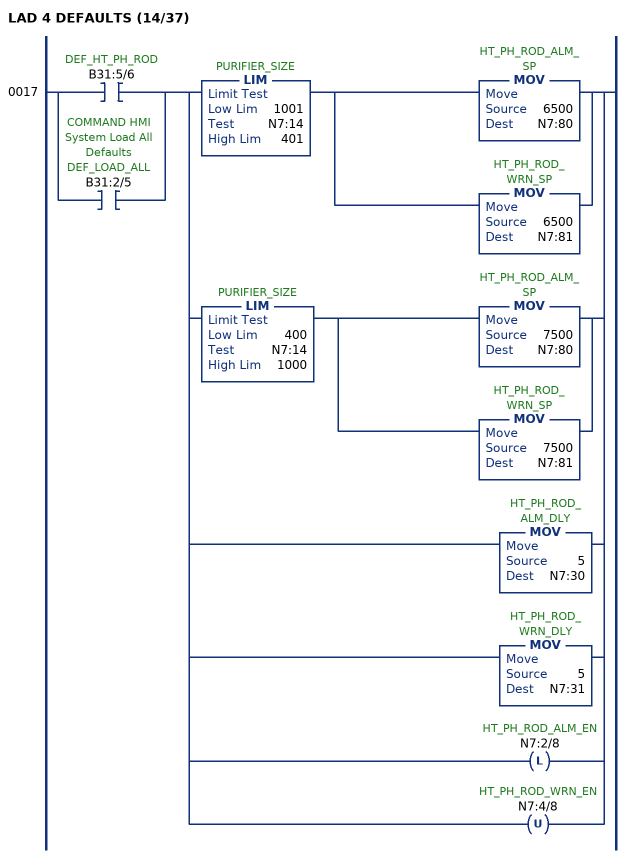
% Rung: 17 %
SOR BST XIC B31:5/6 NXB XIC B31:2/5 BND BST LIM 1001 N7:14 401 BST MOV 6500 N7:80 NXB MOV 6500 N7:81 BND NXB LIM 400 N7:14 1000 BST MOV 7500 N7:80 NXB MOV 7500 N7:81 BND NXB MOV 5 N7:30 NXB MOV 5 N7:31 NXB OTL N7:2/8 NXB OTU N7:4/8 BND EOR
%   B31:5/6  DEF_HT_PH_ROD %
%   B31:2/5  DEF_LOAD_ALL  "COMMAND HMI System Load All Defaults" %
%   N7:14  PURIFIER_SIZE %
%   N7:80  HT_PH_ROD_ALM_SP %
%   N7:81  HT_PH_ROD_WRN_SP %
%   N7:30  HT_PH_ROD_ALM_DLY %
%   N7:31  HT_PH_ROD_WRN_DLY %
%   N7:2/8  HT_PH_ROD_ALM_EN %
%   N7:4/8  HT_PH_ROD_WRN_EN %

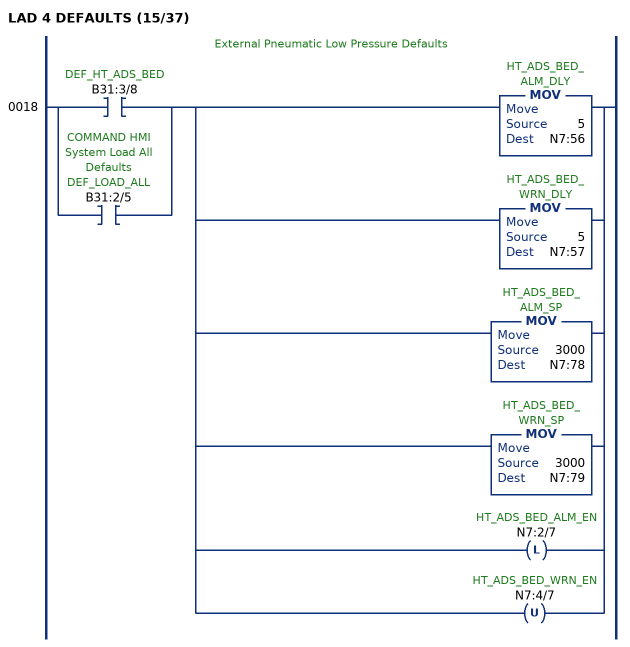
% Rung: 18 %
% External Pneumatic Low Pressure Defaults %
SOR BST XIC B31:3/8 NXB XIC B31:2/5 BND BST MOV 5 N7:56 NXB MOV 5 N7:57 NXB MOV 3000 N7:78 NXB MOV 3000 N7:79 NXB OTL N7:2/7 NXB OTU N7:4/7 BND EOR
%   B31:3/8  DEF_HT_ADS_BED %
%   B31:2/5  DEF_LOAD_ALL  "COMMAND HMI System Load All Defaults" %
%   N7:56  HT_ADS_BED_ALM_DLY %
%   N7:57  HT_ADS_BED_WRN_DLY %
%   N7:78  HT_ADS_BED_ALM_SP %
%   N7:79  HT_ADS_BED_WRN_SP %
%   N7:2/7  HT_ADS_BED_ALM_EN %
%   N7:4/7  HT_ADS_BED_WRN_EN %

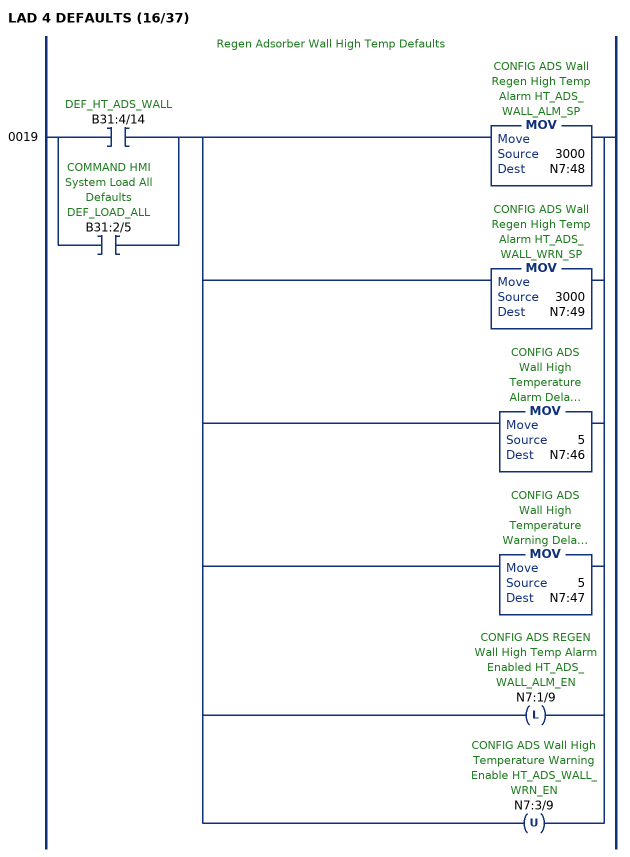
% Rung: 19 %
% Regen Adsorber Wall High Temp Defaults %
SOR BST XIC B31:4/14 NXB XIC B31:2/5 BND BST BST MOV 3000 N7:48 NXB MOV 3000 N7:49 BND NXB MOV 5 N7:46 NXB MOV 5 N7:47 NXB OTL N7:1/9 NXB OTU N7:3/9 BND EOR
%   B31:4/14  DEF_HT_ADS_WALL %
%   B31:2/5  DEF_LOAD_ALL  "COMMAND HMI System Load All Defaults" %
%   N7:48  HT_ADS_WALL_ALM_SP  "CONFIG ADS Wall Regen High Temp Alarm" %
%   N7:49  HT_ADS_WALL_WRN_SP  "CONFIG ADS Wall Regen High Temp Alarm" %
%   N7:46  HT_ADS_WALL_ALM_DLY  "CONFIG ADS Wall High Temperature Alarm Delay" %
%   N7:47  HT_ADS_WALL_WRN_DLY  "CONFIG ADS Wall High Temperature Warning Delay" %
%   N7:1/9  HT_ADS_WALL_ALM_EN  "CONFIG ADS REGEN Wall High Temp Alarm Enabled" %
%   N7:3/9  HT_ADS_WALL_WRN_EN  "CONFIG ADS Wall High Temperature Warning Enable" %

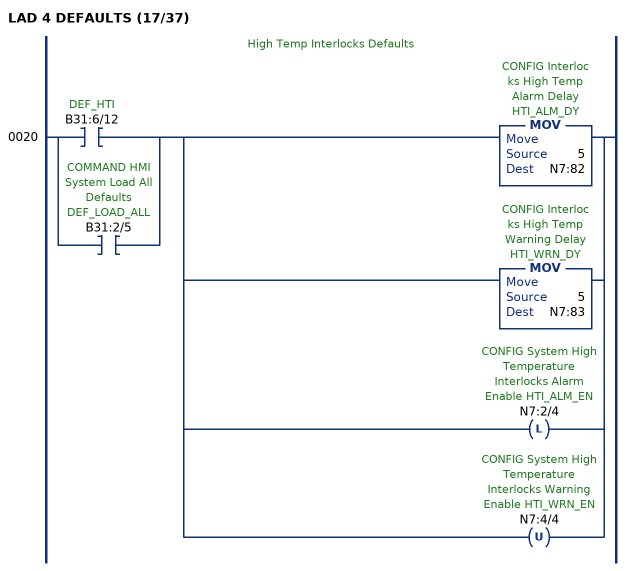
% Rung: 20 %
% High Temp Interlocks Defaults %
SOR BST XIC B31:6/12 NXB XIC B31:2/5 BND BST MOV 5 N7:82 NXB MOV 5 N7:83 NXB OTL N7:2/4 NXB OTU N7:4/4 BND EOR
%   B31:6/12  DEF_HTI %
%   B31:2/5  DEF_LOAD_ALL  "COMMAND HMI System Load All Defaults" %
%   N7:82  HTI_ALM_DY  "CONFIG Interlocks High Temp Alarm Delay" %
%   N7:83  HTI_WRN_DY  "CONFIG Interlocks High Temp Warning Delay" %
%   N7:2/4  HTI_ALM_EN  "CONFIG System High Temperature Interlocks Alarm Enable" %
%   N7:4/4  HTI_WRN_EN  "CONFIG System High Temperature Interlocks Warning Enable" %

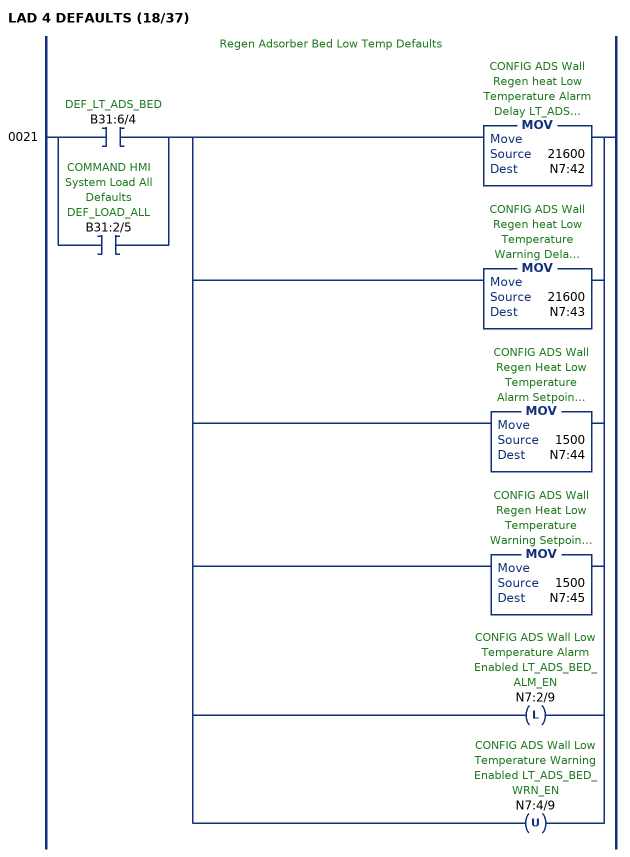
% Rung: 21 %
% Regen Adsorber Bed Low Temp Defaults %
SOR BST XIC B31:6/4 NXB XIC B31:2/5 BND BST MOV 21600 N7:42 NXB MOV 21600 N7:43 NXB MOV 1500 N7:44 NXB MOV 1500 N7:45 NXB OTL N7:2/9 NXB OTU N7:4/9 BND EOR
%   B31:6/4  DEF_LT_ADS_BED %
%   B31:2/5  DEF_LOAD_ALL  "COMMAND HMI System Load All Defaults" %
%   N7:42  LT_ADS_BED_ALM_DLY  "CONFIG ADS Wall Regen heat Low Temperature Alarm Delay" %
%   N7:43  LT_ADS_BED_WRN_DLY  "CONFIG ADS Wall Regen heat Low Temperature Warning Delay" %
%   N7:44  LT_ADS_BED_ALM_SP  "CONFIG ADS Wall Regen Heat Low Temperature Alarm Setpoint" %
%   N7:45  LT_ADS_BED_WRN_SP  "CONFIG ADS Wall Regen Heat Low Temperature Warning Setpoint" %
%   N7:2/9  LT_ADS_BED_ALM_EN  "CONFIG ADS Wall Low Temperature Alarm Enabled" %
%   N7:4/9  LT_ADS_BED_WRN_EN  "CONFIG ADS Wall Low Temperature Warning Enabled" %

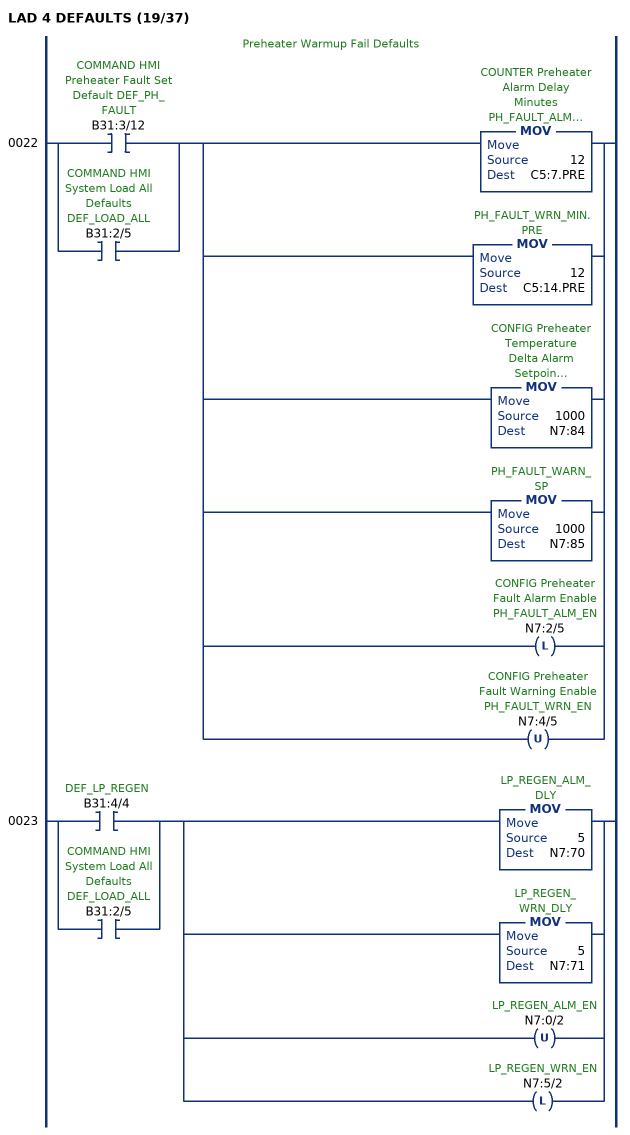
% Rung: 22 %
% Preheater Warmup Fail Defaults %
SOR BST XIC B31:3/12 NXB XIC B31:2/5 BND BST MOV 12 C5:7.PRE NXB MOV 12 C5:14.PRE NXB MOV 1000 N7:84 NXB MOV 1000 N7:85 NXB OTL N7:2/5 NXB OTU N7:4/5 BND EOR
%   B31:3/12  DEF_PH_FAULT  "COMMAND HMI Preheater Fault Set Default" %
%   B31:2/5  DEF_LOAD_ALL  "COMMAND HMI System Load All Defaults" %
%   C5:7  PH_FAULT_ALM_MIN  "COUNTER Preheater Alarm Delay Minutes" %
%   C5:14  PH_FAULT_WRN_MIN %
%   N7:84  PH_FAULT_ALARM_SP  "CONFIG Preheater Temperature Delta Alarm Setpoint" %
%   N7:85  PH_FAULT_WARN_SP %
%   N7:2/5  PH_FAULT_ALM_EN  "CONFIG Preheater Fault Alarm Enable" %
%   N7:4/5  PH_FAULT_WRN_EN  "CONFIG Preheater Fault Warning Enable" %
% Rung: 23 %
SOR BST XIC B31:4/4 NXB XIC B31:2/5 BND BST MOV 5 N7:70 NXB MOV 5 N7:71 NXB OTU N7:0/2 NXB OTL N7:5/2 BND EOR
%   B31:4/4  DEF_LP_REGEN %
%   B31:2/5  DEF_LOAD_ALL  "COMMAND HMI System Load All Defaults" %
%   N7:70  LP_REGEN_ALM_DLY %
%   N7:71  LP_REGEN_WRN_DLY %
%   N7:0/2  LP_REGEN_ALM_EN %
%   N7:5/2  LP_REGEN_WRN_EN %

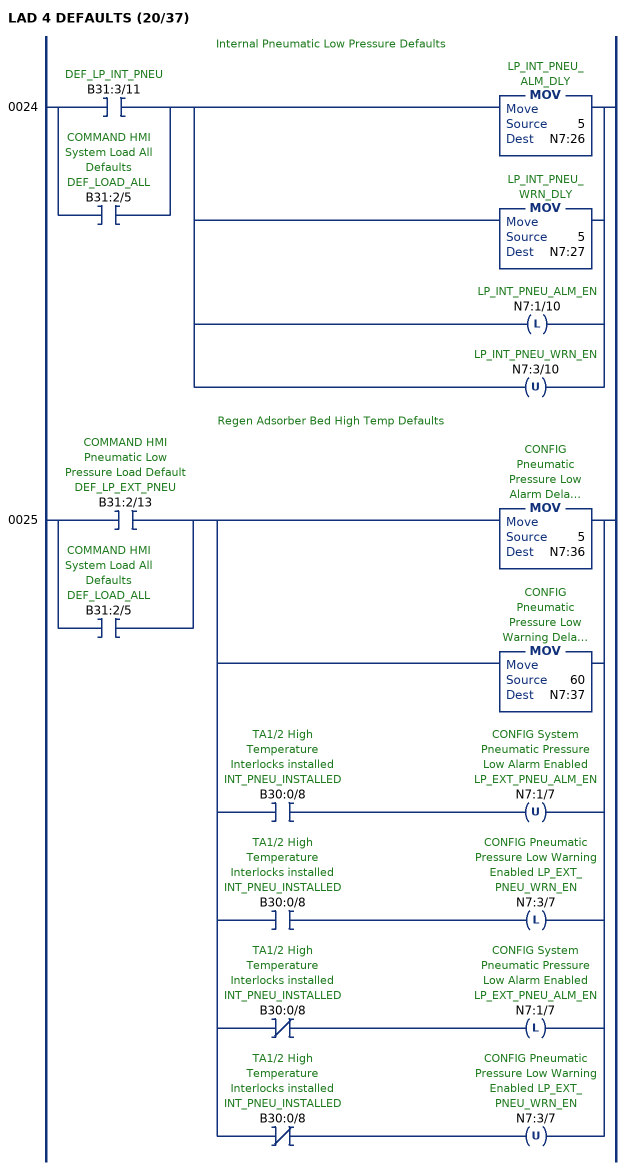
% Rung: 24 %
% Internal Pneumatic Low Pressure Defaults %
SOR BST XIC B31:3/11 NXB XIC B31:2/5 BND BST MOV 5 N7:26 NXB MOV 5 N7:27 NXB OTL N7:1/10 NXB OTU N7:3/10 BND EOR
%   B31:3/11  DEF_LP_INT_PNEU %
%   B31:2/5  DEF_LOAD_ALL  "COMMAND HMI System Load All Defaults" %
%   N7:26  LP_INT_PNEU_ALM_DLY %
%   N7:27  LP_INT_PNEU_WRN_DLY %
%   N7:1/10  LP_INT_PNEU_ALM_EN %
%   N7:3/10  LP_INT_PNEU_WRN_EN %
% Rung: 25 %
% Regen Adsorber Bed High Temp Defaults %
SOR BST XIC B31:2/13 NXB XIC B31:2/5 BND BST MOV 5 N7:36 NXB MOV 60 N7:37 NXB XIC B30:0/8 OTU N7:1/7 NXB XIC B30:0/8 OTL N7:3/7 NXB XIO B30:0/8 OTL N7:1/7 NXB XIO B30:0/8 OTU N7:3/7 BND EOR
%   B31:2/13  DEF_LP_EXT_PNEU  "COMMAND HMI Pneumatic Low Pressure Load Default" %
%   B31:2/5  DEF_LOAD_ALL  "COMMAND HMI System Load All Defaults" %
%   N7:36  LP_EXT_PNEU_ALM_DLY  "CONFIG Pneumatic Pressure Low Alarm Delay" %
%   N7:37  LP_EXT_PNEU_WRN_DLY  "CONFIG Pneumatic Pressure Low Warning Delay" %
%   B30:0/8  INT_PNEU_INSTALLED  "TA1/2 High Temperature Interlocks installed" %
%   N7:1/7  LP_EXT_PNEU_ALM_EN  "CONFIG System Pneumatic Pressure Low Alarm Enabled" %
%   N7:3/7  LP_EXT_PNEU_WRN_EN  "CONFIG Pneumatic Pressure Low Warning Enabled" %

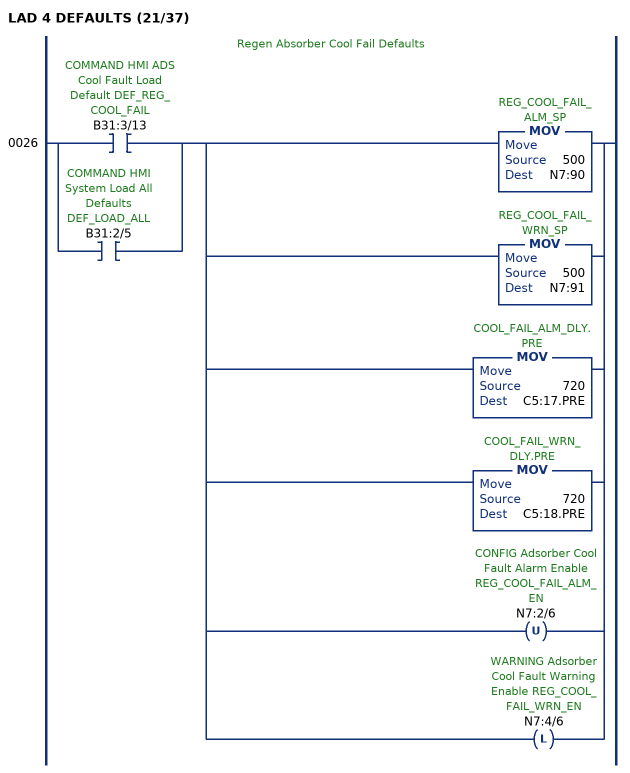
% Rung: 26 %
% Regen Absorber Cool Fail Defaults %
SOR BST XIC B31:3/13 NXB XIC B31:2/5 BND BST MOV 500 N7:90 NXB MOV 500 N7:91 NXB MOV 720 C5:17.PRE NXB MOV 720 C5:18.PRE NXB OTU N7:2/6 NXB OTL N7:4/6 BND EOR
%   B31:3/13  DEF_REG_COOL_FAIL  "COMMAND HMI ADS Cool Fault Load Default" %
%   B31:2/5  DEF_LOAD_ALL  "COMMAND HMI System Load All Defaults" %
%   N7:90  REG_COOL_FAIL_ALM_SP %
%   N7:91  REG_COOL_FAIL_WRN_SP %
%   C5:17  COOL_FAIL_ALM_DLY %
%   C5:18  COOL_FAIL_WRN_DLY %
%   N7:2/6  REG_COOL_FAIL_ALM_EN  "CONFIG Adsorber Cool Fault Alarm Enable" %
%   N7:4/6  REG_COOL_FAIL_WRN_EN  "WARNING Adsorber Cool Fault Warning Enable" %

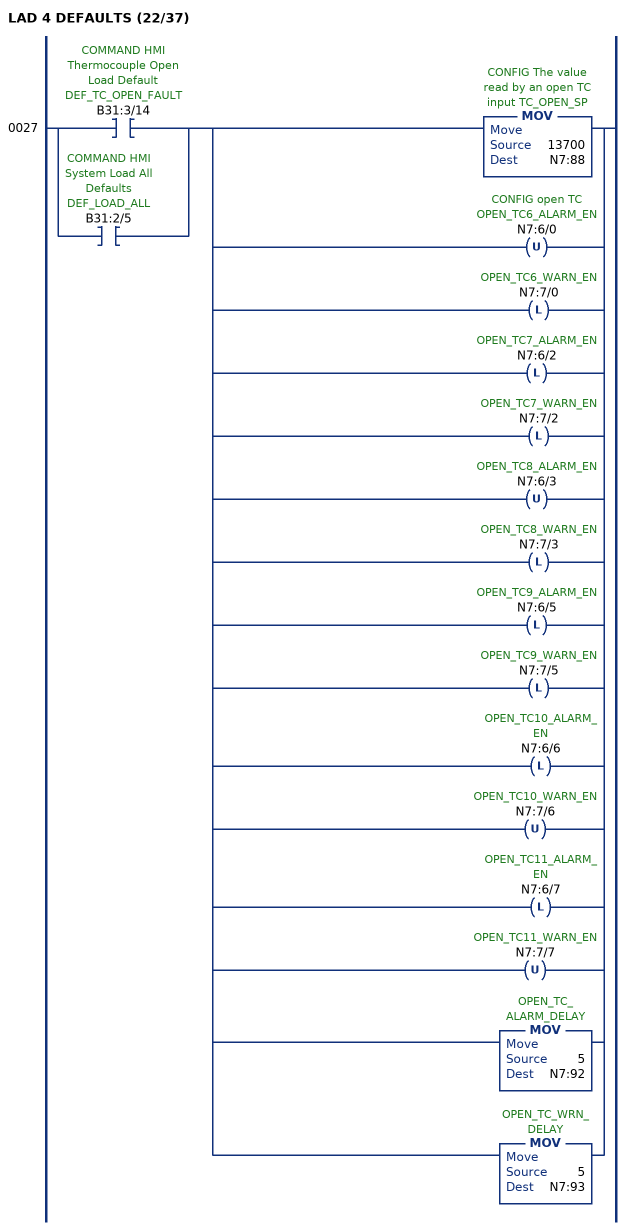
% Rung: 27 %
SOR BST XIC B31:3/14 NXB XIC B31:2/5 BND BST MOV 13700 N7:88 NXB OTU N7:6/0 NXB OTL N7:7/0 NXB OTL N7:6/2 NXB OTL N7:7/2 NXB OTU N7:6/3 NXB OTL N7:7/3 NXB OTL N7:6/5 NXB OTL N7:7/5 NXB OTL N7:6/6 NXB OTU N7:7/6 NXB OTL N7:6/7 NXB BST OTU N7:7/7 NXB BST MOV 5 N7:92 NXB MOV 5 N7:93 BND BND BND EOR
%   B31:3/14  DEF_TC_OPEN_FAULT  "COMMAND HMI Thermocouple Open Load Default" %
%   B31:2/5  DEF_LOAD_ALL  "COMMAND HMI System Load All Defaults" %
%   N7:88  TC_OPEN_SP  "CONFIG The value read by an open TC input" %
%   N7:6/0  OPEN_TC6_ALARM_EN  "CONFIG open TC" %
%   N7:7/0  OPEN_TC6_WARN_EN %
%   N7:6/2  OPEN_TC7_ALARM_EN %
%   N7:7/2  OPEN_TC7_WARN_EN %
%   N7:6/3  OPEN_TC8_ALARM_EN %
%   N7:7/3  OPEN_TC8_WARN_EN %
%   N7:6/5  OPEN_TC9_ALARM_EN %
%   N7:7/5  OPEN_TC9_WARN_EN %
%   N7:6/6  OPEN_TC10_ALARM_EN %
%   N7:7/6  OPEN_TC10_WARN_EN %
%   N7:6/7  OPEN_TC11_ALARM_EN %
%   N7:7/7  OPEN_TC11_WARN_EN %
%   N7:92  OPEN_TC_ALARM_DELAY %
%   N7:93  OPEN_TC_WRN_DELAY %

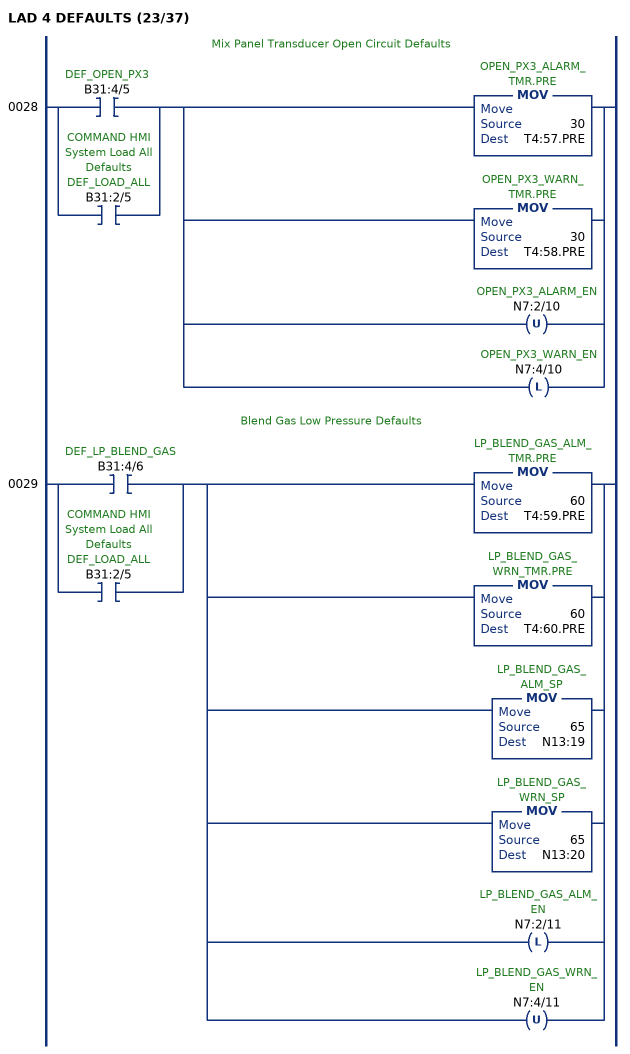
% Rung: 28 %
% Mix Panel Transducer Open Circuit Defaults %
SOR BST XIC B31:4/5 NXB XIC B31:2/5 BND BST MOV 30 T4:57.PRE NXB MOV 30 T4:58.PRE NXB OTU N7:2/10 NXB OTL N7:4/10 BND EOR
%   B31:4/5  DEF_OPEN_PX3 %
%   B31:2/5  DEF_LOAD_ALL  "COMMAND HMI System Load All Defaults" %
%   T4:57  OPEN_PX3_ALARM_TMR %
%   T4:58  OPEN_PX3_WARN_TMR %
%   N7:2/10  OPEN_PX3_ALARM_EN %
%   N7:4/10  OPEN_PX3_WARN_EN %
% Rung: 29 %
% Blend Gas Low Pressure Defaults %
SOR BST XIC B31:4/6 NXB XIC B31:2/5 BND BST MOV 60 T4:59.PRE NXB MOV 60 T4:60.PRE NXB MOV 65 N13:19 NXB MOV 65 N13:20 NXB OTL N7:2/11 NXB OTU N7:4/11 BND EOR
%   B31:4/6  DEF_LP_BLEND_GAS %
%   B31:2/5  DEF_LOAD_ALL  "COMMAND HMI System Load All Defaults" %
%   T4:59  LP_BLEND_GAS_ALM_TMR %
%   T4:60  LP_BLEND_GAS_WRN_TMR %
%   N13:19  LP_BLEND_GAS_ALM_SP %
%   N13:20  LP_BLEND_GAS_WRN_SP %
%   N7:2/11  LP_BLEND_GAS_ALM_EN %
%   N7:4/11  LP_BLEND_GAS_WRN_EN %

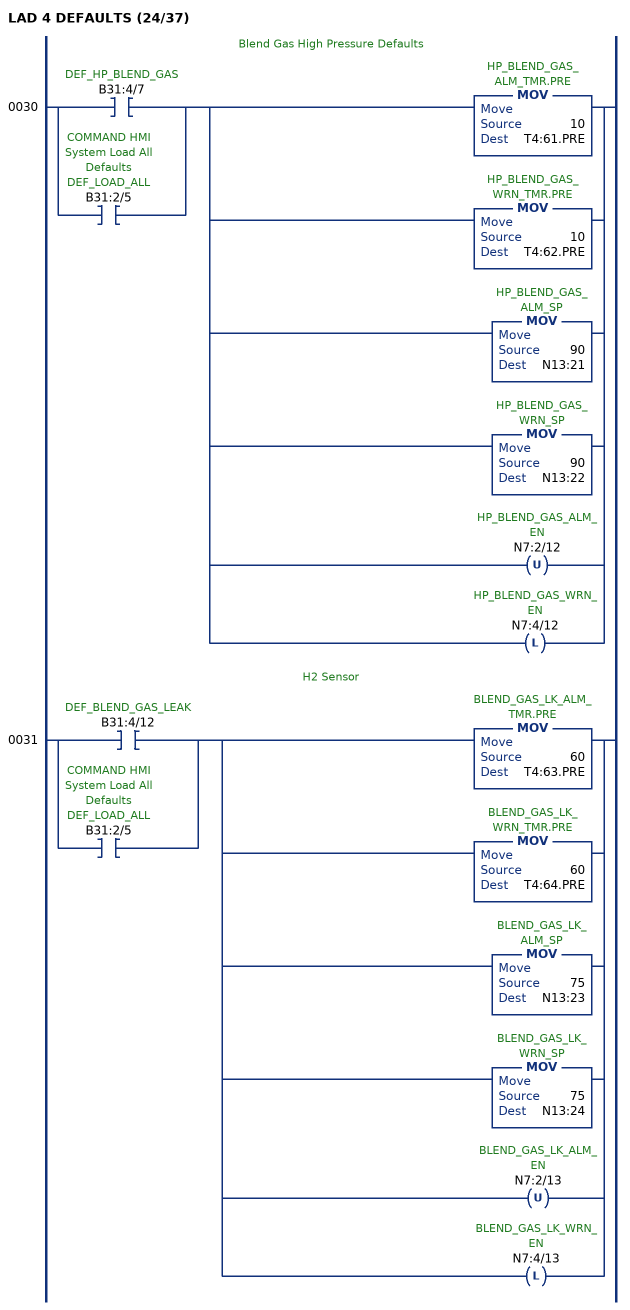
% Rung: 30 %
% Blend Gas High Pressure Defaults %
SOR BST XIC B31:4/7 NXB XIC B31:2/5 BND BST MOV 10 T4:61.PRE NXB MOV 10 T4:62.PRE NXB MOV 90 N13:21 NXB MOV 90 N13:22 NXB OTU N7:2/12 NXB OTL N7:4/12 BND EOR
%   B31:4/7  DEF_HP_BLEND_GAS %
%   B31:2/5  DEF_LOAD_ALL  "COMMAND HMI System Load All Defaults" %
%   T4:61  HP_BLEND_GAS_ALM_TMR %
%   T4:62  HP_BLEND_GAS_WRN_TMR %
%   N13:21  HP_BLEND_GAS_ALM_SP %
%   N13:22  HP_BLEND_GAS_WRN_SP %
%   N7:2/12  HP_BLEND_GAS_ALM_EN %
%   N7:4/12  HP_BLEND_GAS_WRN_EN %
% Rung: 31 %
% H2 Sensor %
SOR BST XIC B31:4/12 NXB XIC B31:2/5 BND BST MOV 60 T4:63.PRE NXB MOV 60 T4:64.PRE NXB MOV 75 N13:23 NXB MOV 75 N13:24 NXB OTU N7:2/13 NXB OTL N7:4/13 BND EOR
%   B31:4/12  DEF_BLEND_GAS_LEAK %
%   B31:2/5  DEF_LOAD_ALL  "COMMAND HMI System Load All Defaults" %
%   T4:63  BLEND_GAS_LK_ALM_TMR %
%   T4:64  BLEND_GAS_LK_WRN_TMR %
%   N13:23  BLEND_GAS_LK_ALM_SP %
%   N13:24  BLEND_GAS_LK_WRN_SP %
%   N7:2/13  BLEND_GAS_LK_ALM_EN %
%   N7:4/13  BLEND_GAS_LK_WRN_EN %

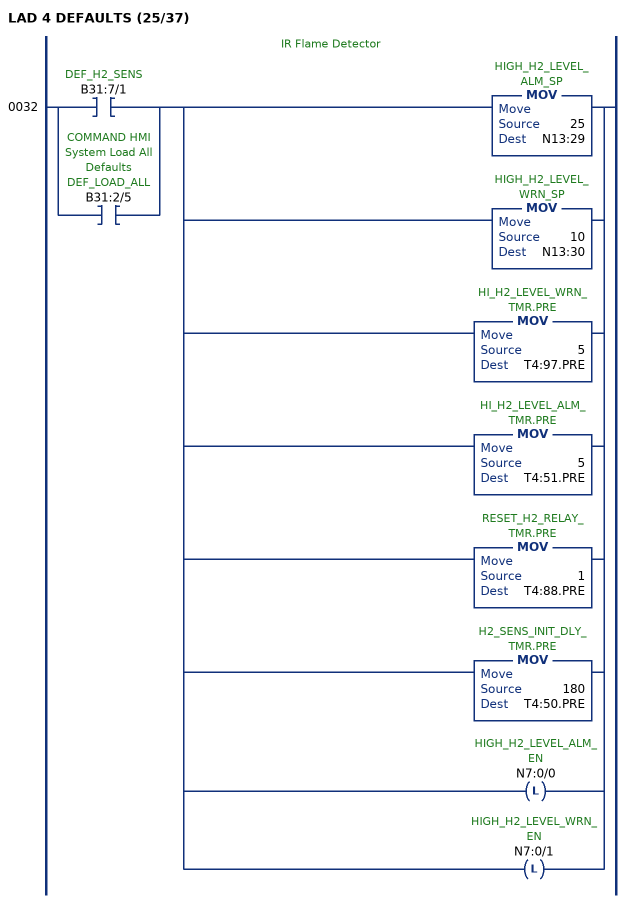
% Rung: 32 %
% IR Flame Detector %
SOR BST XIC B31:7/1 NXB XIC B31:2/5 BND BST MOV 25 N13:29 NXB MOV 10 N13:30 NXB MOV 5 T4:97.PRE NXB MOV 5 T4:51.PRE NXB MOV 1 T4:88.PRE NXB MOV 180 T4:50.PRE NXB OTL N7:0/0 NXB OTL N7:0/1 BND EOR
%   B31:7/1  DEF_H2_SENS %
%   B31:2/5  DEF_LOAD_ALL  "COMMAND HMI System Load All Defaults" %
%   N13:29  HIGH_H2_LEVEL_ALM_SP %
%   N13:30  HIGH_H2_LEVEL_WRN_SP %
%   T4:97  HI_H2_LEVEL_WRN_TMR %
%   T4:51  HI_H2_LEVEL_ALM_TMR %
%   T4:88  RESET_H2_RELAY_TMR %
%   T4:50  H2_SENS_INIT_DLY_TMR %
%   N7:0/0  HIGH_H2_LEVEL_ALM_EN %
%   N7:0/1  HIGH_H2_LEVEL_WRN_EN %

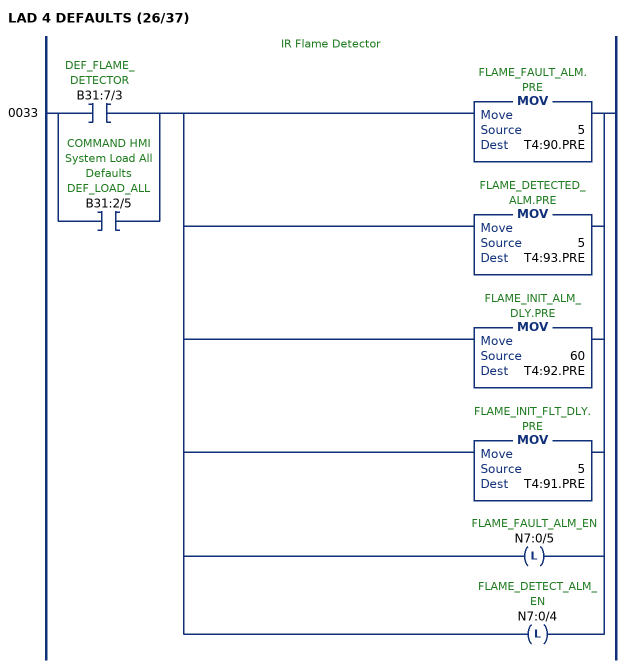
% Rung: 33 %
% IR Flame Detector %
SOR BST XIC B31:7/3 NXB XIC B31:2/5 BND BST MOV 5 T4:90.PRE NXB MOV 5 T4:93.PRE NXB MOV 60 T4:92.PRE NXB MOV 5 T4:91.PRE NXB OTL N7:0/5 NXB OTL N7:0/4 BND EOR
%   B31:7/3  DEF_FLAME_DETECTOR %
%   B31:2/5  DEF_LOAD_ALL  "COMMAND HMI System Load All Defaults" %
%   T4:90  FLAME_FAULT_ALM %
%   T4:93  FLAME_DETECTED_ALM %
%   T4:92  FLAME_INIT_ALM_DLY %
%   T4:91  FLAME_INIT_FLT_DLY %
%   N7:0/5  FLAME_FAULT_ALM_EN %
%   N7:0/4  FLAME_DETECT_ALM_EN %

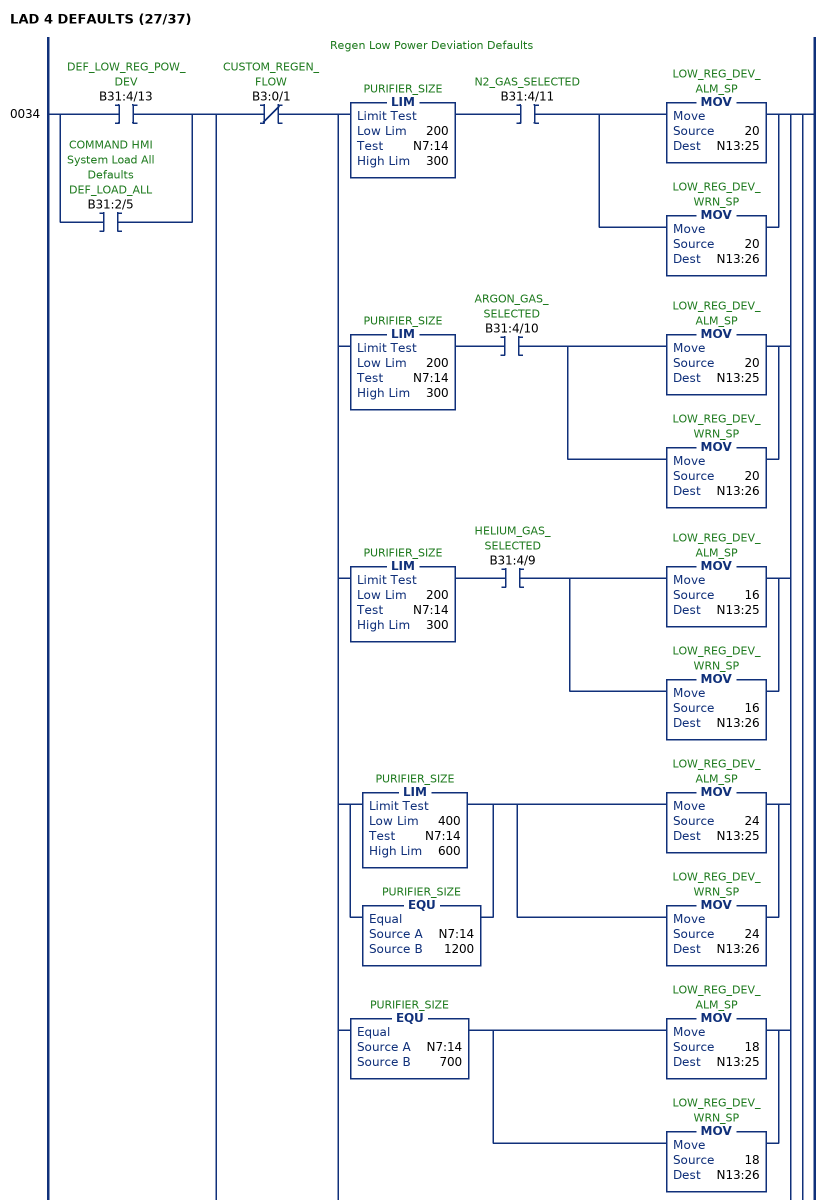

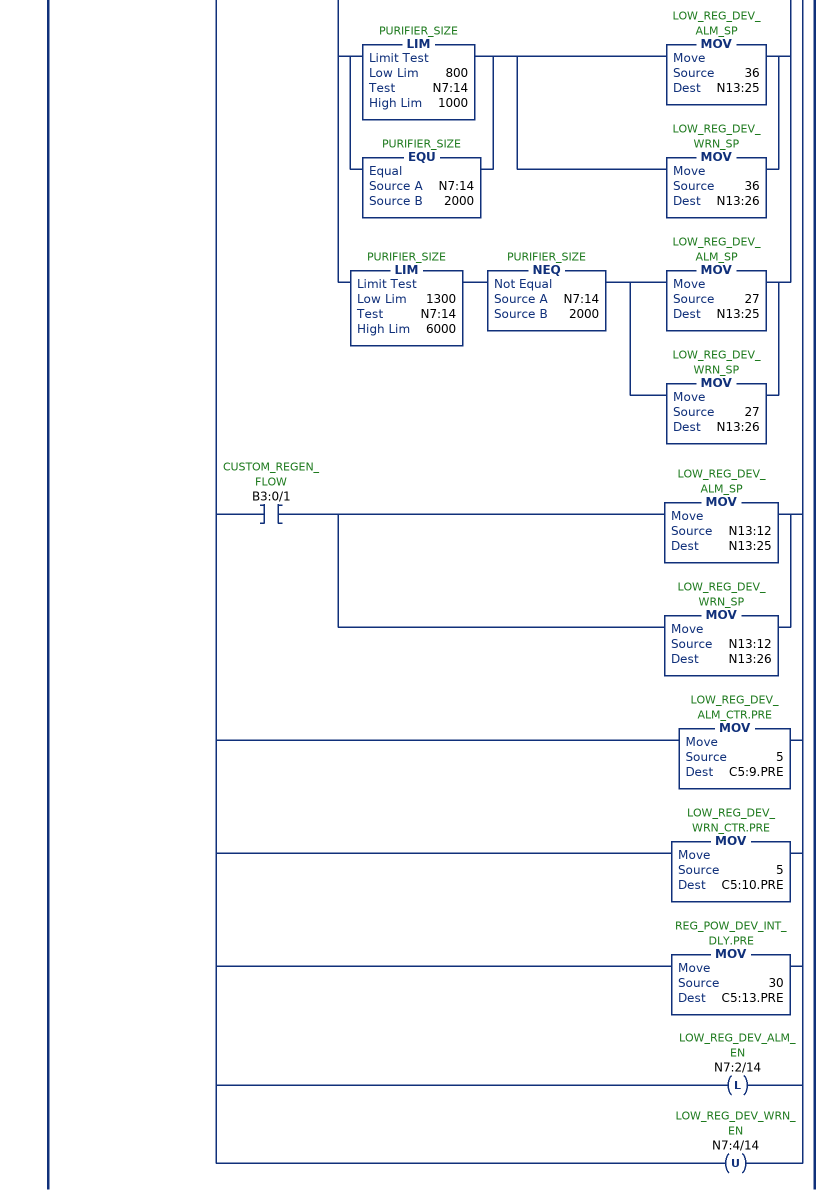
% Rung: 34 %
% Regen Low Power Deviation Defaults %
SOR BST XIC B31:4/13 NXB XIC B31:2/5 BND BST XIO B3:0/1 BST LIM 200 N7:14 300 XIC B31:4/11 BST MOV 20 N13:25 NXB MOV 20 N13:26 BND NXB LIM 200 N7:14 300 XIC B31:4/10 BST MOV 20 N13:25 NXB MOV 20 N13:26 BND NXB LIM 200 N7:14 300 XIC B31:4/9 BST MOV 16 N13:25 NXB MOV 16 N13:26 BND NXB BST LIM 400 N7:14 600 NXB EQU N7:14 1200 BND BST MOV 24 N13:25 NXB MOV 24 N13:26 BND NXB EQU N7:14 700 BST MOV 18 N13:25 NXB MOV 18 N13:26 BND NXB BST LIM 800 N7:14 1000 NXB EQU N7:14 2000 BND BST MOV 36 N13:25 NXB MOV 36 N13:26 BND NXB LIM 1300 N7:14 6000 NEQ N7:14 2000 BST MOV 27 N13:25 NXB MOV 27 N13:26 BND BND NXB XIC B3:0/1 BST MOV N13:12 N13:25 NXB MOV N13:12 N13:26 BND NXB MOV 5 C5:9.PRE NXB MOV 5 C5:10.PRE NXB MOV 30 C5:13.PRE NXB OTL N7:2/14 NXB OTU N7:4/14 BND EOR
%   B31:4/13  DEF_LOW_REG_POW_DEV %
%   B31:2/5  DEF_LOAD_ALL  "COMMAND HMI System Load All Defaults" %
%   B3:0/1  CUSTOM_REGEN_FLOW %
%   N7:14  PURIFIER_SIZE %
%   B31:4/11  N2_GAS_SELECTED %
%   N13:25  LOW_REG_DEV_ALM_SP %
%   N13:26  LOW_REG_DEV_WRN_SP %
%   B31:4/10  ARGON_GAS_SELECTED %
%   B31:4/9  HELIUM_GAS_SELECTED %
%   N13:12  CUST_LOW_REG_DEV_SP %
%   C5:9  LOW_REG_DEV_ALM_CTR %
%   C5:10  LOW_REG_DEV_WRN_CTR %
%   C5:13  REG_POW_DEV_INT_DLY %
%   N7:2/14  LOW_REG_DEV_ALM_EN %
%   N7:4/14  LOW_REG_DEV_WRN_EN %

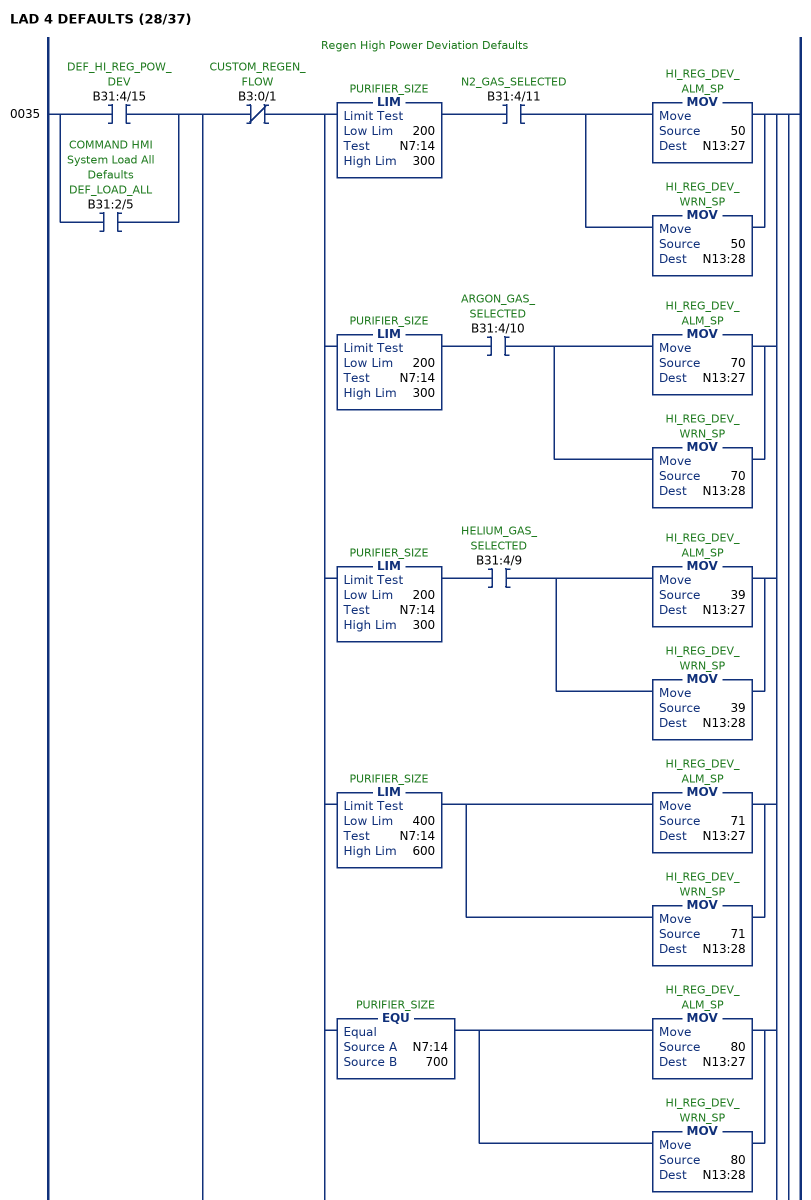

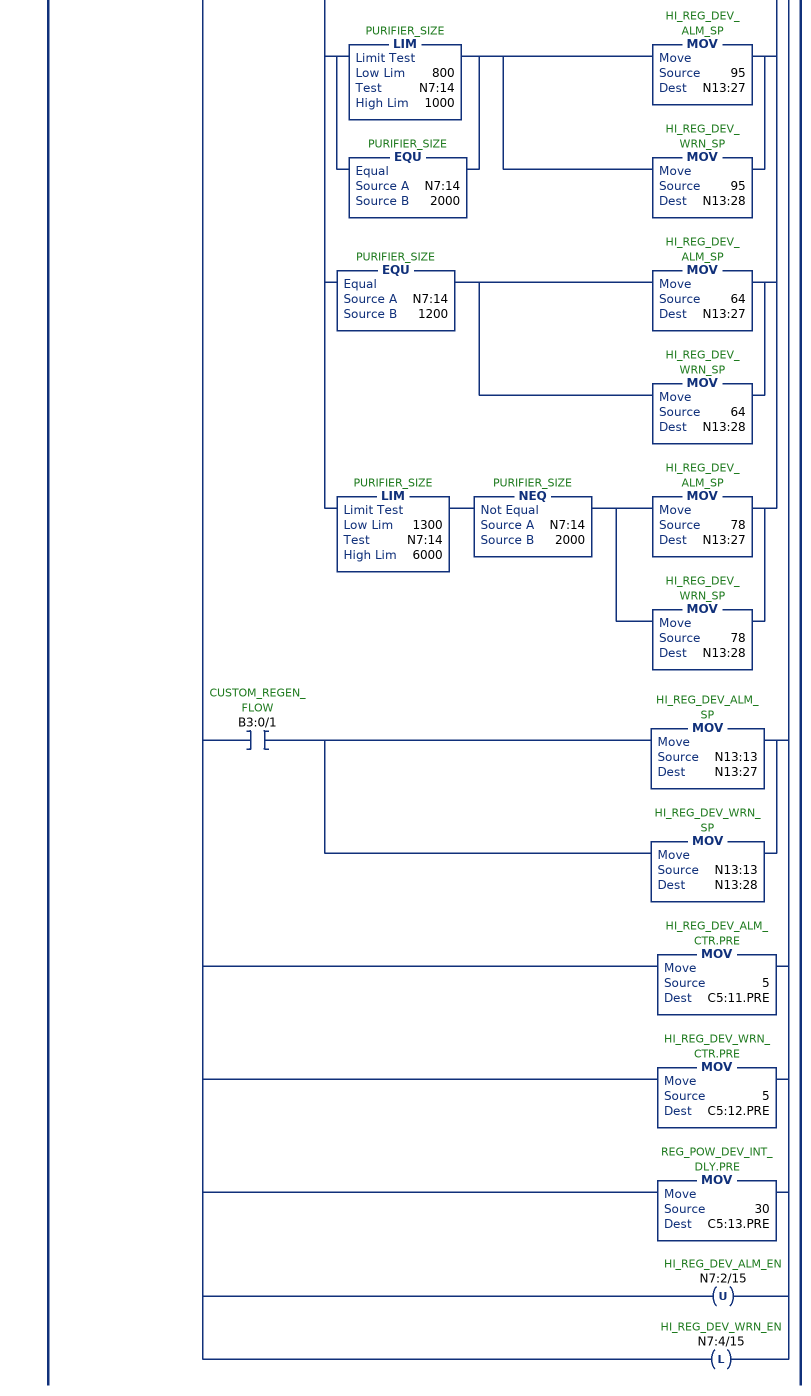
% Rung: 35 %
% Regen High Power Deviation Defaults %
SOR BST XIC B31:4/15 NXB XIC B31:2/5 BND BST XIO B3:0/1 BST LIM 200 N7:14 300 XIC B31:4/11 BST MOV 50 N13:27 NXB MOV 50 N13:28 BND NXB LIM 200 N7:14 300 XIC B31:4/10 BST MOV 70 N13:27 NXB MOV 70 N13:28 BND NXB LIM 200 N7:14 300 XIC B31:4/9 BST MOV 39 N13:27 NXB MOV 39 N13:28 BND NXB LIM 400 N7:14 600 BST MOV 71 N13:27 NXB MOV 71 N13:28 BND NXB EQU N7:14 700 BST MOV 80 N13:27 NXB MOV 80 N13:28 BND NXB BST LIM 800 N7:14 1000 NXB EQU N7:14 2000 BND BST MOV 95 N13:27 NXB MOV 95 N13:28 BND NXB EQU N7:14 1200 BST MOV 64 N13:27 NXB MOV 64 N13:28 BND NXB LIM 1300 N7:14 6000 NEQ N7:14 2000 BST MOV 78 N13:27 NXB MOV 78 N13:28 BND BND NXB XIC B3:0/1 BST MOV N13:13 N13:27 NXB MOV N13:13 N13:28 BND NXB MOV 5 C5:11.PRE NXB MOV 5 C5:12.PRE NXB MOV 30 C5:13.PRE NXB OTU N7:2/15 NXB OTL N7:4/15 BND EOR
%   B31:4/15  DEF_HI_REG_POW_DEV %
%   B31:2/5  DEF_LOAD_ALL  "COMMAND HMI System Load All Defaults" %
%   B3:0/1  CUSTOM_REGEN_FLOW %
%   N7:14  PURIFIER_SIZE %
%   B31:4/11  N2_GAS_SELECTED %
%   N13:27  HI_REG_DEV_ALM_SP %
%   N13:28  HI_REG_DEV_WRN_SP %
%   B31:4/10  ARGON_GAS_SELECTED %
%   B31:4/9  HELIUM_GAS_SELECTED %
%   N13:13  CUST_HI_REG_DEV_SP %
%   C5:11  HI_REG_DEV_ALM_CTR %
%   C5:12  HI_REG_DEV_WRN_CTR %
%   C5:13  REG_POW_DEV_INT_DLY %
%   N7:2/15  HI_REG_DEV_ALM_EN %
%   N7:4/15  HI_REG_DEV_WRN_EN %

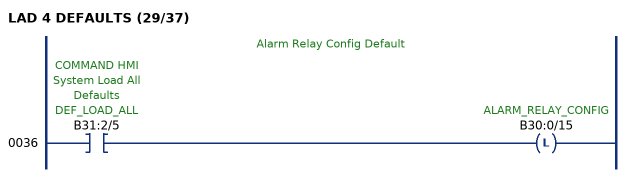
% Rung: 36 %
% Alarm Relay Config Default %
SOR XIC B31:2/5 OTL B30:0/15 EOR
%   B31:2/5  DEF_LOAD_ALL  "COMMAND HMI System Load All Defaults" %
%   B30:0/15  ALARM_RELAY_CONFIG %

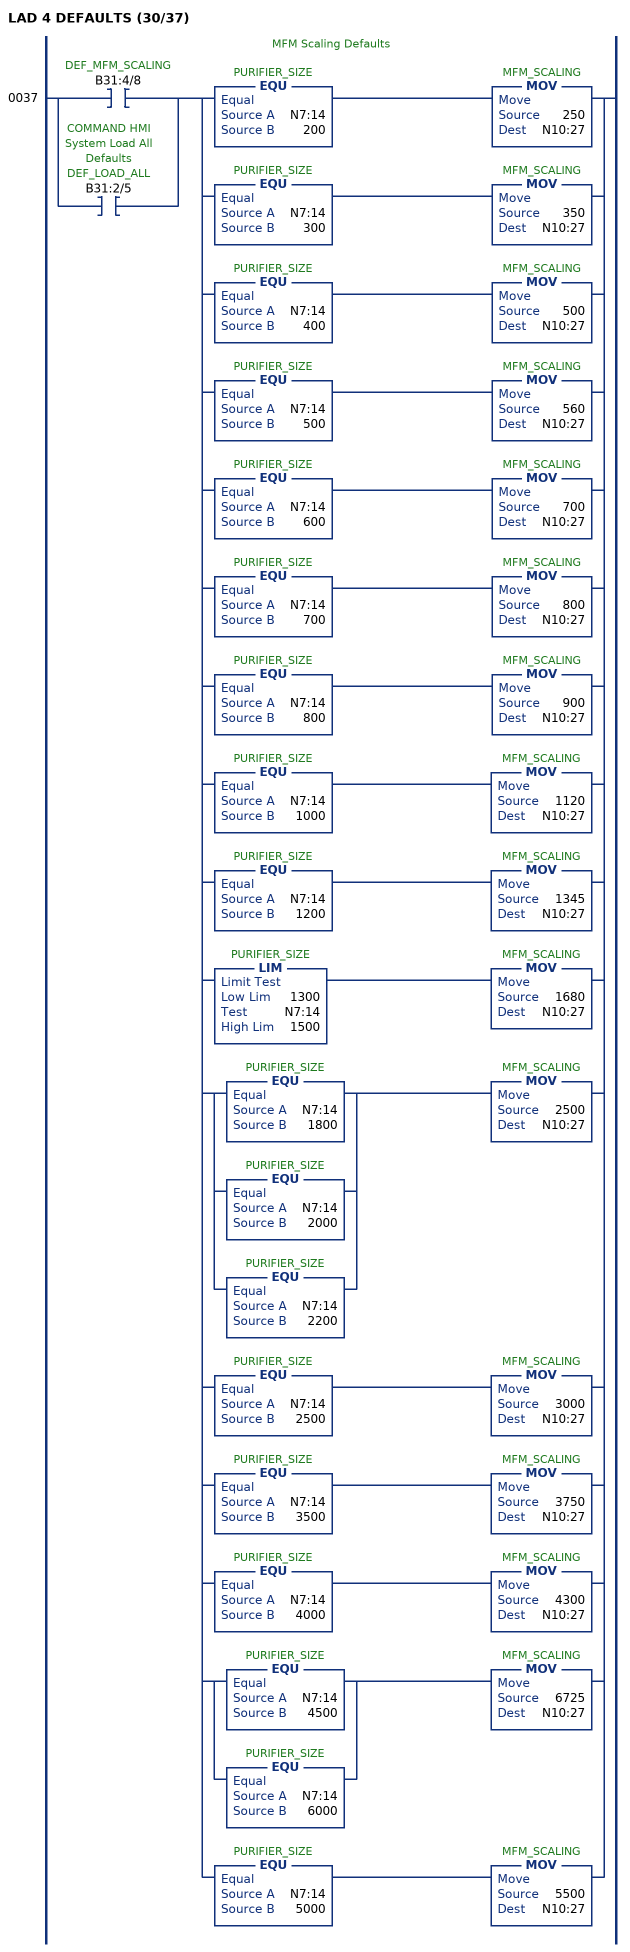
% Rung: 37 %
% MFM Scaling Defaults %
SOR BST XIC B31:4/8 NXB XIC B31:2/5 BND BST EQU N7:14 200 MOV 250 N10:27 NXB EQU N7:14 300 MOV 350 N10:27 NXB EQU N7:14 400 MOV 500 N10:27 NXB EQU N7:14 500 MOV 560 N10:27 NXB EQU N7:14 600 MOV 700 N10:27 NXB EQU N7:14 700 MOV 800 N10:27 NXB EQU N7:14 800 MOV 900 N10:27 NXB EQU N7:14 1000 MOV 1120 N10:27 NXB EQU N7:14 1200 MOV 1345 N10:27 NXB LIM 1300 N7:14 1500 MOV 1680 N10:27 NXB BST EQU N7:14 1800 NXB EQU N7:14 2000 NXB EQU N7:14 2200 BND MOV 2500 N10:27 NXB EQU N7:14 2500 MOV 3000 N10:27 NXB EQU N7:14 3500 MOV 3750 N10:27 NXB EQU N7:14 4000 MOV 4300 N10:27 NXB BST EQU N7:14 4500 NXB EQU N7:14 6000 BND MOV 6725 N10:27 NXB EQU N7:14 5000 MOV 5500 N10:27 BND EOR
%   B31:4/8  DEF_MFM_SCALING %
%   B31:2/5  DEF_LOAD_ALL  "COMMAND HMI System Load All Defaults" %
%   N7:14  PURIFIER_SIZE %
%   N10:27  MFM_SCALING %

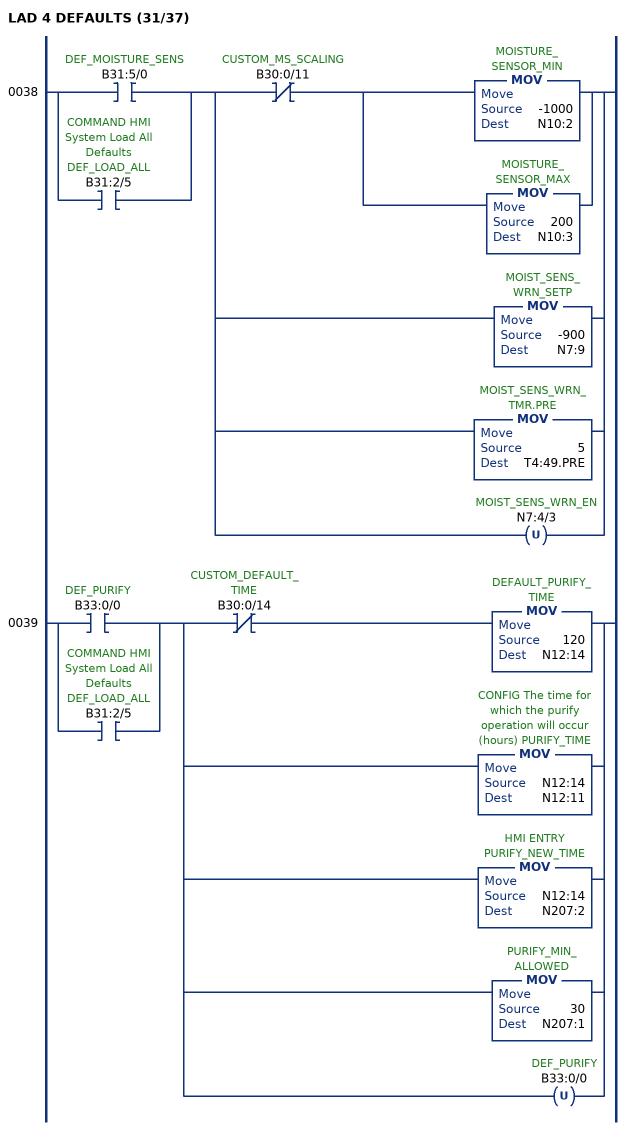
% Rung: 38 %
SOR BST XIC B31:5/0 NXB XIC B31:2/5 BND BST XIO B30:0/11 BST MOV -1000 N10:2 NXB MOV 200 N10:3 BND NXB MOV -900 N7:9 NXB MOV 5 T4:49.PRE NXB OTU N7:4/3 BND EOR
%   B31:5/0  DEF_MOISTURE_SENS %
%   B31:2/5  DEF_LOAD_ALL  "COMMAND HMI System Load All Defaults" %
%   B30:0/11  CUSTOM_MS_SCALING %
%   N10:2  MOISTURE_SENSOR_MIN %
%   N10:3  MOISTURE_SENSOR_MAX %
%   N7:9  MOIST_SENS_WRN_SETP %
%   T4:49  MOIST_SENS_WRN_TMR %
%   N7:4/3  MOIST_SENS_WRN_EN %
% Rung: 39 %
SOR BST XIC B33:0/0 NXB XIC B31:2/5 BND BST XIO B30:0/14 MOV 120 N12:14 NXB MOV N12:14 N12:11 NXB MOV N12:14 N207:2 NXB MOV 30 N207:1 NXB OTU B33:0/0 BND EOR
%   B33:0/0  DEF_PURIFY %
%   B31:2/5  DEF_LOAD_ALL  "COMMAND HMI System Load All Defaults" %
%   B30:0/14  CUSTOM_DEFAULT_TIME %
%   N12:14  DEFAULT_PURIFY_TIME %
%   N12:11  PURIFY_TIME  "CONFIG The time for which the purify operation will occur (hours)" %
%   N207:2  PURIFY_NEW_TIME  "HMI ENTRY" %
%   N207:1  PURIFY_MIN_ALLOWED %

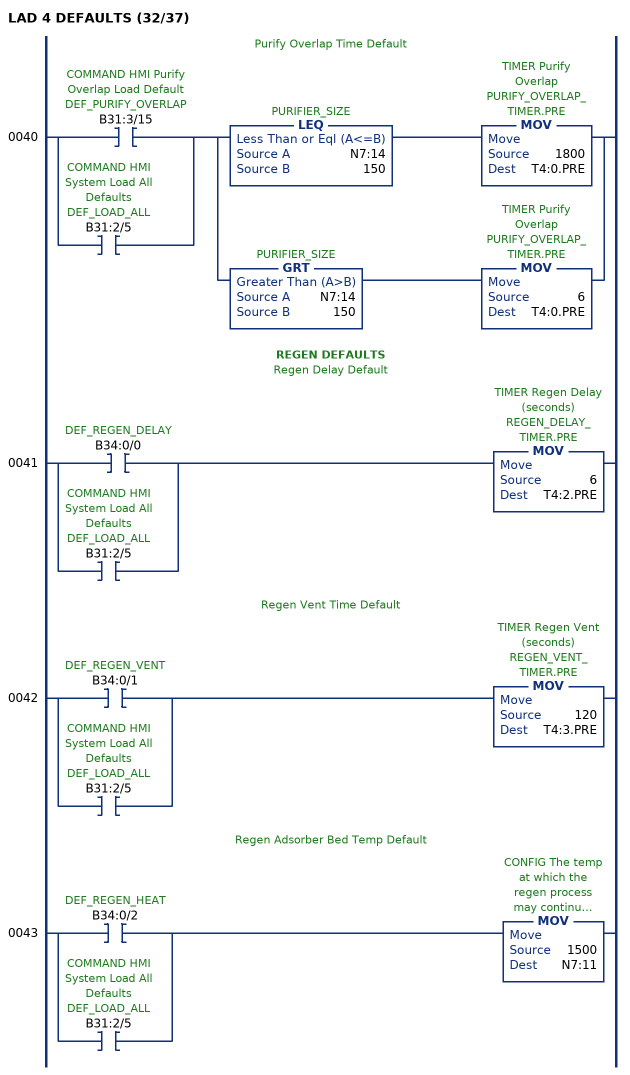
% Rung: 40 %
% Purify Overlap Time Default %
SOR BST XIC B31:3/15 NXB XIC B31:2/5 BND BST LEQ N7:14 150 MOV 1800 T4:0.PRE NXB GRT N7:14 150 MOV 6 T4:0.PRE BND EOR
%   B31:3/15  DEF_PURIFY_OVERLAP  "COMMAND HMI Purify Overlap Load Default" %
%   B31:2/5  DEF_LOAD_ALL  "COMMAND HMI System Load All Defaults" %
%   N7:14  PURIFIER_SIZE %
%   T4:0  PURIFY_OVERLAP_TIMER  "TIMER Purify Overlap" %
% Rung: 41 %
% TITLE: REGEN DEFAULTS %
% Regen Delay Default %
SOR BST XIC B34:0/0 NXB XIC B31:2/5 BND MOV 6 T4:2.PRE EOR
%   B34:0/0  DEF_REGEN_DELAY %
%   B31:2/5  DEF_LOAD_ALL  "COMMAND HMI System Load All Defaults" %
%   T4:2  REGEN_DELAY_TIMER  "TIMER Regen Delay (seconds)" %
% Rung: 42 %
% Regen Vent Time Default %
SOR BST XIC B34:0/1 NXB XIC B31:2/5 BND MOV 120 T4:3.PRE EOR
%   B34:0/1  DEF_REGEN_VENT %
%   B31:2/5  DEF_LOAD_ALL  "COMMAND HMI System Load All Defaults" %
%   T4:3  REGEN_VENT_TIMER  "TIMER Regen Vent (seconds)" %
% Rung: 43 %
% Regen Adsorber Bed Temp Default %
SOR BST XIC B34:0/2 NXB XIC B31:2/5 BND MOV 1500 N7:11 EOR
%   B34:0/2  DEF_REGEN_HEAT %
%   B31:2/5  DEF_LOAD_ALL  "COMMAND HMI System Load All Defaults" %
%   N7:11  ADS_BED_TEMP_HIGH  "CONFIG The temp at which the regen process may continue" %

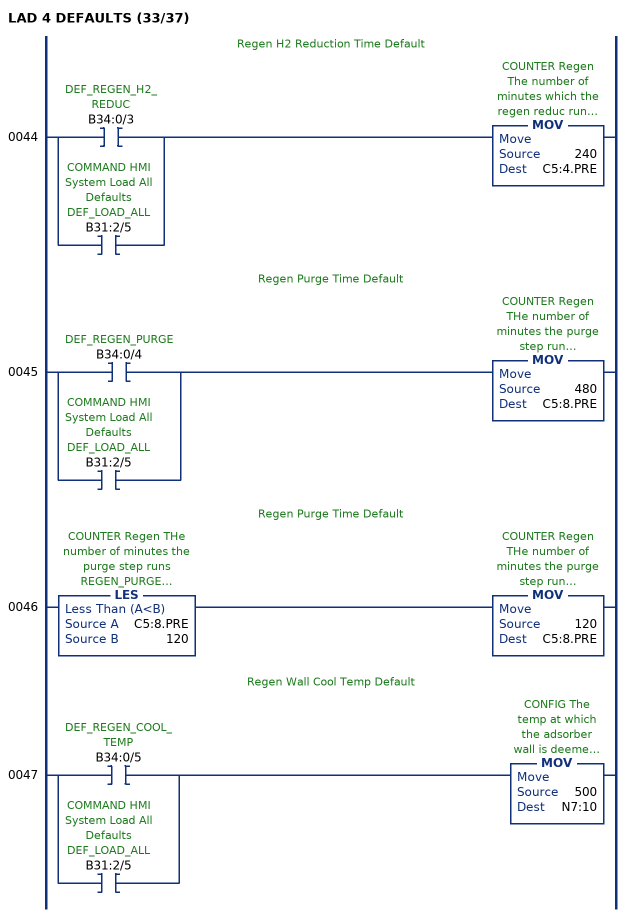
% Rung: 44 %
% Regen H2 Reduction Time Default %
SOR BST XIC B34:0/3 NXB XIC B31:2/5 BND MOV 240 C5:4.PRE EOR
%   B34:0/3  DEF_REGEN_H2_REDUC %
%   B31:2/5  DEF_LOAD_ALL  "COMMAND HMI System Load All Defaults" %
%   C5:4  REGEN_REDUC_MINUTE  "COUNTER Regen The number of minutes which the regen reduc runs" %
% Rung: 45 %
% Regen Purge Time Default %
SOR BST XIC B34:0/4 NXB XIC B31:2/5 BND MOV 480 C5:8.PRE EOR
%   B34:0/4  DEF_REGEN_PURGE %
%   B31:2/5  DEF_LOAD_ALL  "COMMAND HMI System Load All Defaults" %
%   C5:8  REGEN_PURGE_MINUTES  "COUNTER Regen THe number of minutes the purge step runs" %
% Rung: 46 %
% Regen Purge Time Default %
SOR LES C5:8.PRE 120 MOV 120 C5:8.PRE EOR
%   C5:8  REGEN_PURGE_MINUTES  "COUNTER Regen THe number of minutes the purge step runs" %
% Rung: 47 %
% Regen Wall Cool Temp Default %
SOR BST XIC B34:0/5 NXB XIC B31:2/5 BND MOV 500 N7:10 EOR
%   B34:0/5  DEF_REGEN_COOL_TEMP %
%   B31:2/5  DEF_LOAD_ALL  "COMMAND HMI System Load All Defaults" %
%   N7:10  ADS_WALL_TEMP_COOL  "CONFIG The temp at which the adsorber wall is deemed to be cool enough to purify" %

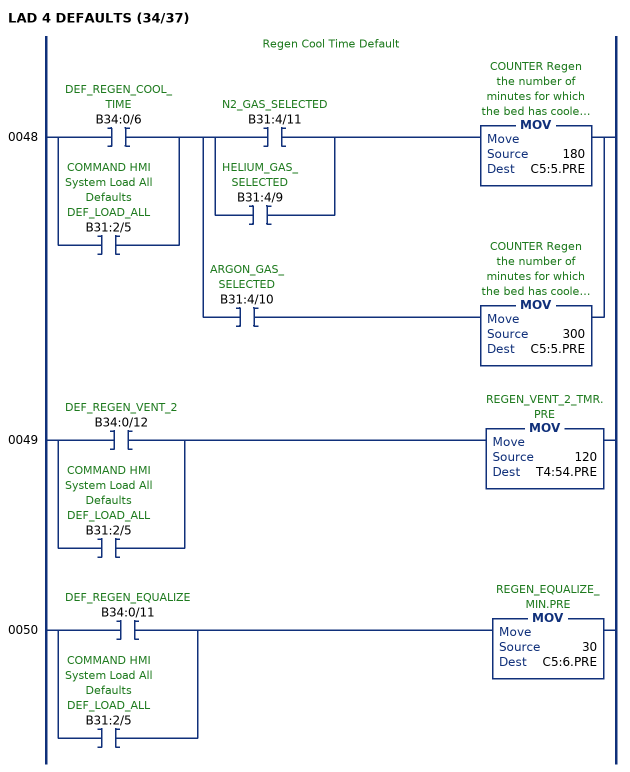
% Rung: 48 %
% Regen Cool Time Default %
SOR BST XIC B34:0/6 NXB XIC B31:2/5 BND BST BST XIC B31:4/11 NXB XIC B31:4/9 BND MOV 180 C5:5.PRE NXB XIC B31:4/10 MOV 300 C5:5.PRE BND EOR
%   B34:0/6  DEF_REGEN_COOL_TIME %
%   B31:2/5  DEF_LOAD_ALL  "COMMAND HMI System Load All Defaults" %
%   B31:4/11  N2_GAS_SELECTED %
%   B31:4/9  HELIUM_GAS_SELECTED %
%   C5:5  REGEN_COOL_MINUTE  "COUNTER Regen the number of minutes for which the bed has cooled" %
%   B31:4/10  ARGON_GAS_SELECTED %
% Rung: 49 %
SOR BST XIC B34:0/12 NXB XIC B31:2/5 BND MOV 120 T4:54.PRE EOR
%   B34:0/12  DEF_REGEN_VENT_2 %
%   B31:2/5  DEF_LOAD_ALL  "COMMAND HMI System Load All Defaults" %
%   T4:54  REGEN_VENT_2_TMR %
% Rung: 50 %
SOR BST XIC B34:0/11 NXB XIC B31:2/5 BND MOV 30 C5:6.PRE EOR
%   B34:0/11  DEF_REGEN_EQUALIZE %
%   B31:2/5  DEF_LOAD_ALL  "COMMAND HMI System Load All Defaults" %
%   C5:6  REGEN_EQUALIZE_MIN %

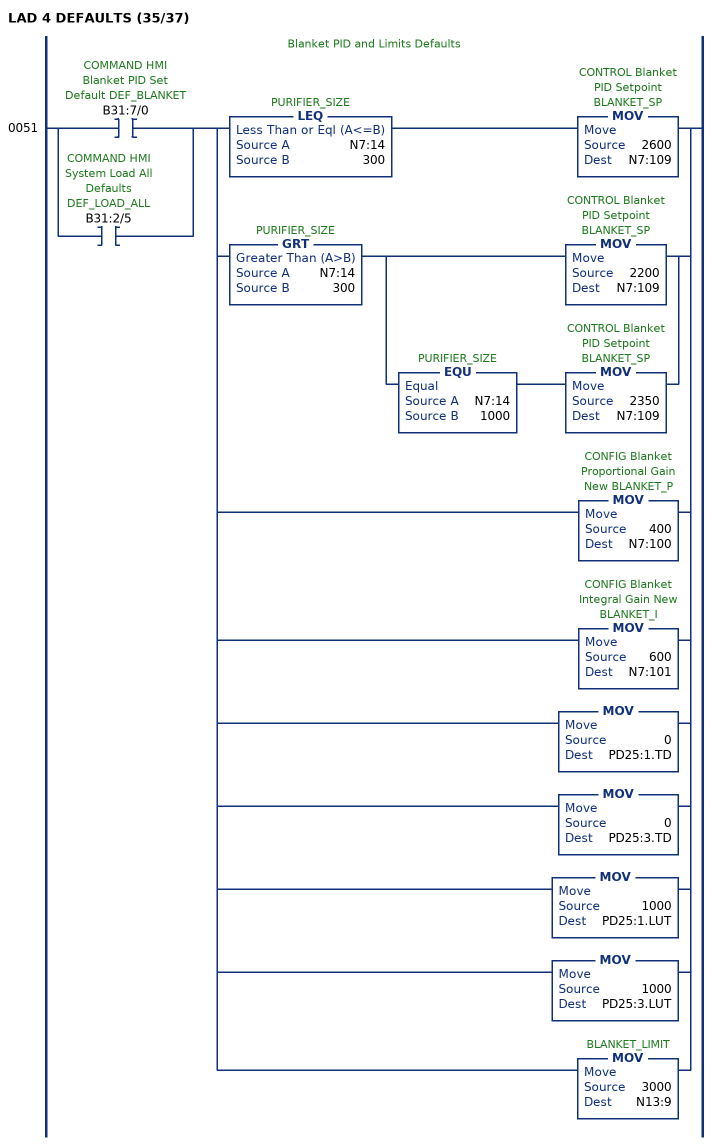
% Rung: 51 %
% Blanket PID and Limits Defaults %
SOR BST XIC B31:7/0 NXB XIC B31:2/5 BND BST LEQ N7:14 300 MOV 2600 N7:109 NXB GRT N7:14 300 BST MOV 2200 N7:109 NXB EQU N7:14 1000 MOV 2350 N7:109 BND NXB MOV 400 N7:100 NXB MOV 600 N7:101 NXB MOV 0 PD25:1.TD NXB MOV 0 PD25:3.TD NXB MOV 1000 PD25:1.LUT NXB MOV 1000 PD25:3.LUT NXB MOV 3000 N13:9 BND EOR
%   B31:7/0  DEF_BLANKET  "COMMAND HMI Blanket PID Set Default" %
%   B31:2/5  DEF_LOAD_ALL  "COMMAND HMI System Load All Defaults" %
%   N7:14  PURIFIER_SIZE %
%   N7:109  BLANKET_SP  "CONTROL Blanket PID Setpoint" %
%   N7:100  BLANKET_P  "CONFIG Blanket Proportional Gain New" %
%   N7:101  BLANKET_I  "CONFIG Blanket Integral Gain New" %
%   N13:9  BLANKET_LIMIT %

